// TwinCAT 3 PLC project PLC
// ProgramVersion: 3.1.4026.19
// CompilerDefines: VISU_USEPROPERTYINFO
// libraries:
//   Tc2_Standard, * (Beckhoff Automation GmbH)
//   Tc2_System, * (Beckhoff Automation GmbH)
//   VisuSymbols, 4.5.0.0 (System)
// project tree:
//   / GlobalTextList.TcGTLO, PlcTask.TcTTO, Visualization Manager.TcVMO (not stored)
//   POUs/ MAIN.TcPOU
//   VISUs/ Visualization.TcVIS

CONFIGURATION PLC
    RESOURCE PLC ON TwinCAT3
        TASK PlcTask(INTERVAL := T#10ms, PRIORITY := 20);
        PROGRAM MAIN WITH PlcTask : MAIN;
    END_RESOURCE
END_CONFIGURATION

// ---- POUs/MAIN.TcPOU
PROGRAM MAIN
VAR
	bStartButton : BOOL;
	bStopButton: BOOL;
	bLimitSwitch: BOOL;
	bMotor: BOOL;
END_VAR

IF bStopButton OR bLimitSwitch THEN
    bMotor := FALSE;         
    bStartButton := FALSE;   // <-- Doğru yer burası! (Sadece Stop veya Switch aktifse çalışır)

ELSIF bStartButton THEN
    bMotor := TRUE;          // <-- Buraya bStartButton := FALSE YAZMIYORUZ!
END_IF

END_PROGRAM

// ---- VISUs/Visualization.TcVIS
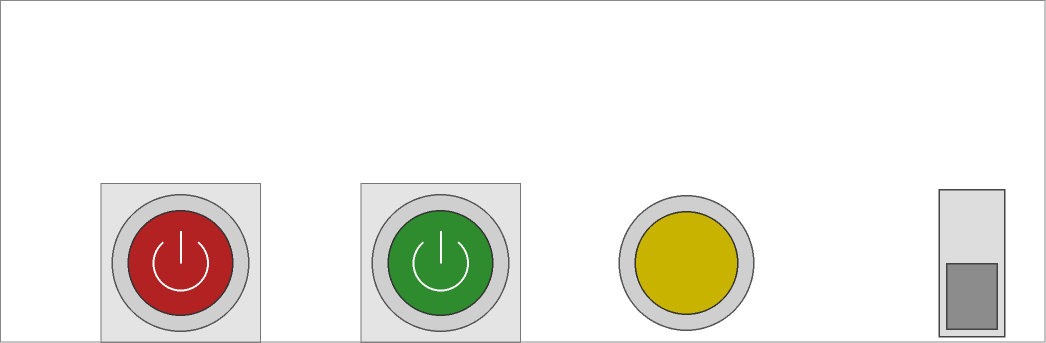
VISUALIZATION Visualization  // 1046x343
    PowerSwitch (83,183 195x160), variable: MAIN.bStopButton, behaviour: TOGGLE, style: Switch-PowerSwitch-Red
    PowerSwitch (343,183 195x160), variable: MAIN.bStartButton, behaviour: TOGGLE, style: Switch-PowerSwitch-Green
    Lamp1 (608,183 157x160), variable: MAIN.bMotor, style: Lamp-Lamp1-Yellow
    DipSwitch (898,183 148x160), variable: MAIN.bLimitSwitch, behaviour: TOGGLE, style: Switch-DipSwitch-Gray
END_VISUALIZATION
